(* PLC project motor_project.project, CODESYS CODESYS V3.5 SP8 Patch 2 *)
(* stored: creationDateTime 2016-04-24T17:57:52.8674236, modificationDateTime 2016-04-24T17:42:05.1952198 *)

CONFIGURATION MyMotor
END_CONFIGURATION
